(* Logix 5000 project; controller PRU vendor 1 type 14 code 107 rev 20.13; software revision 20.01; part 7 of 17 *)
(* tags used below, declared in another part *)
   DRYER : DUAL_SCREW;
   FAULT : DINT[100];
   FAULT_TIMER : TIMER[10000];
   FAULTS_FA1A_IOK : BOOL;   // MODULE FAULTS ARE OK.
   HMI_ALARM_RESET : BOOL;
   Module_ENCL_Fault : DINT;
   Module_ENCL_Iok : BOOL;
   Module_ENCL_Status : DINT;
   Module_ENCR_Fault : DINT;
   Module_ENCR_Iok : BOOL;
   Module_ENCR_Status : DINT;
   Module_LAI1_Fault : DINT;
   Module_LAI1_Iok : BOOL;
   Module_LAI1_Status : DINT;
   Module_LAI2_Fault : DINT;
   Module_LAI2_Iok : BOOL;
   Module_LAI2_Status : DINT;
   Module_LAI3_Fault : DINT;
   Module_LAI3_Iok : BOOL;
   Module_LAI3_Status : DINT;
   Module_LAO1_Fault : DINT;
   Module_LAO1_Iok : BOOL;
   Module_LAO1_Status : DINT;
   Module_LAO2_Fault : DINT;
   Module_LAO2_Iok : BOOL;
   Module_LAO2_Status : DINT;
   Module_LDI1_Fault : DINT;
   Module_LDI1_Iok : BOOL;
   Module_LDI1_Status : DINT;
   Module_LDI2_Fault : DINT;
   Module_LDI2_Iok : BOOL;
   Module_LDI2_Status : DINT;
   Module_LDO1_Fault : DINT;
   Module_LDO1_Iok : BOOL;
   Module_LDO1_Status : DINT;
   Module_LDO2_Fault : DINT;
   Module_LDO2_Iok : BOOL;
   Module_LDO2_Status : DINT;
   Module_LTC1_Fault : DINT;
   Module_LTC1_Iok : BOOL;
   Module_LTC1_Status : DINT;
   Module_LTC2_Fault : DINT;
   Module_LTC2_Iok : BOOL;
   Module_LTC2_Status : DINT;
   Module_LTC3_Fault : DINT;
   Module_LTC3_Iok : BOOL;
   Module_LTC3_Status : DINT;
   Module_LTC4_Fault : DINT;
   Module_LTC4_Iok : BOOL;
   Module_LTC4_Status : DINT;
   TE0101 : REAL;
   TE0102 : REAL;
   TE0103 : REAL;
   TE0104 : REAL;
   TE0105 : REAL;
   TE0106 : REAL;
   TE0107 : REAL;
   TE0108 : REAL;
   TE0109 : REAL;
   TE0110 : REAL;
   TE0111 : REAL;
   TE0112 : REAL;
   TE0113 : REAL;
   TE0114 : REAL;
   TE0115 : REAL;
   TE0116 : REAL;
   TE0117 : REAL;
   TE0118 : REAL;
   TE0119 : REAL;
   TE0120 : REAL;
   TE0121 : REAL;
   TE0122 : REAL;
   TE0123 : REAL;
   TE0124 : REAL;
   TE0125 : REAL;
   TE0126 : REAL;
   TE0127 : REAL;
   TE0128 : REAL;
   TE0129 : REAL;
   TE0130 : REAL;
   TE0201 : REAL;
   TE0202 : REAL;
   THRESHOLD : REAL[9000];
   WARNF_IOK : BOOL;
   WARNG_IOK : BOOL;
   WEIGHT : REAL;
(* MainProgram, continued *)

ROUTINE B00_WARN_F_700_LO_TEMP   (* ladder *)
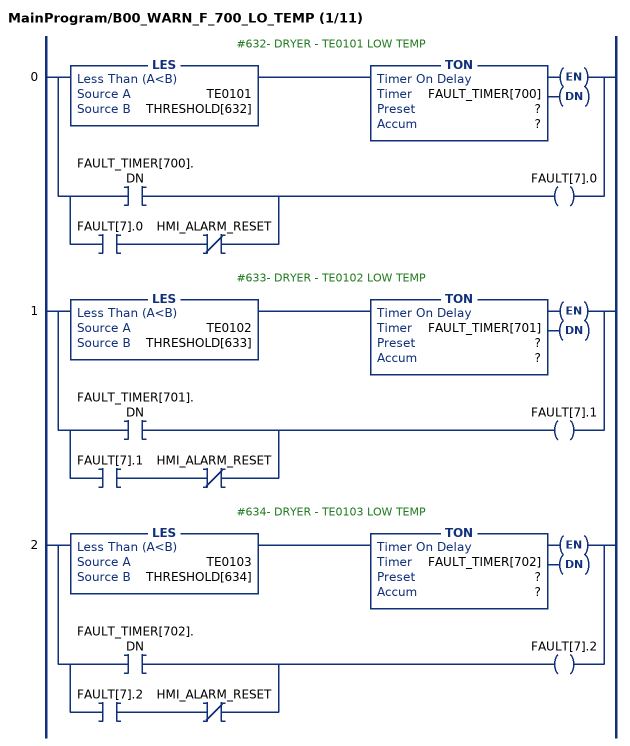
   // #632- DRYER - TE0101 LOW TEMP
   0: [LES(TE0101,THRESHOLD[632]) TON(FAULT_TIMER[700],?,?) ,[XIC(FAULT_TIMER[700].DN) ,XIC(FAULT[7].0) XIO(HMI_ALARM_RESET) ] OTE(FAULT[7].0) ];
   // #633- DRYER - TE0102 LOW TEMP
   1: [LES(TE0102,THRESHOLD[633]) TON(FAULT_TIMER[701],?,?) ,[XIC(FAULT_TIMER[701].DN) ,XIC(FAULT[7].1) XIO(HMI_ALARM_RESET) ] OTE(FAULT[7].1) ];
   // #634- DRYER - TE0103 LOW TEMP
   2: [LES(TE0103,THRESHOLD[634]) TON(FAULT_TIMER[702],?,?) ,[XIC(FAULT_TIMER[702].DN) ,XIC(FAULT[7].2) XIO(HMI_ALARM_RESET) ] OTE(FAULT[7].2) ];
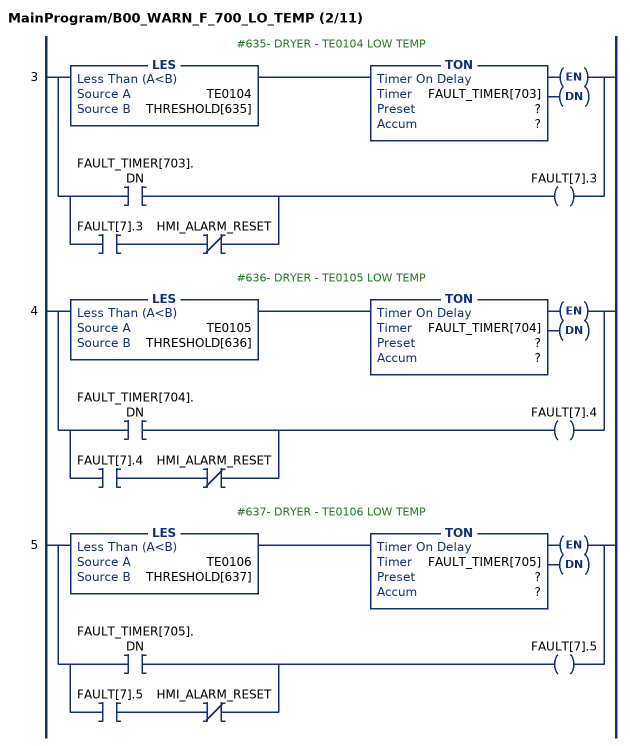
   // #635- DRYER - TE0104 LOW TEMP
   3: [LES(TE0104,THRESHOLD[635]) TON(FAULT_TIMER[703],?,?) ,[XIC(FAULT_TIMER[703].DN) ,XIC(FAULT[7].3) XIO(HMI_ALARM_RESET) ] OTE(FAULT[7].3) ];
   // #636- DRYER - TE0105 LOW TEMP
   4: [LES(TE0105,THRESHOLD[636]) TON(FAULT_TIMER[704],?,?) ,[XIC(FAULT_TIMER[704].DN) ,XIC(FAULT[7].4) XIO(HMI_ALARM_RESET) ] OTE(FAULT[7].4) ];
   // #637- DRYER - TE0106 LOW TEMP
   5: [LES(TE0106,THRESHOLD[637]) TON(FAULT_TIMER[705],?,?) ,[XIC(FAULT_TIMER[705].DN) ,XIC(FAULT[7].5) XIO(HMI_ALARM_RESET) ] OTE(FAULT[7].5) ];
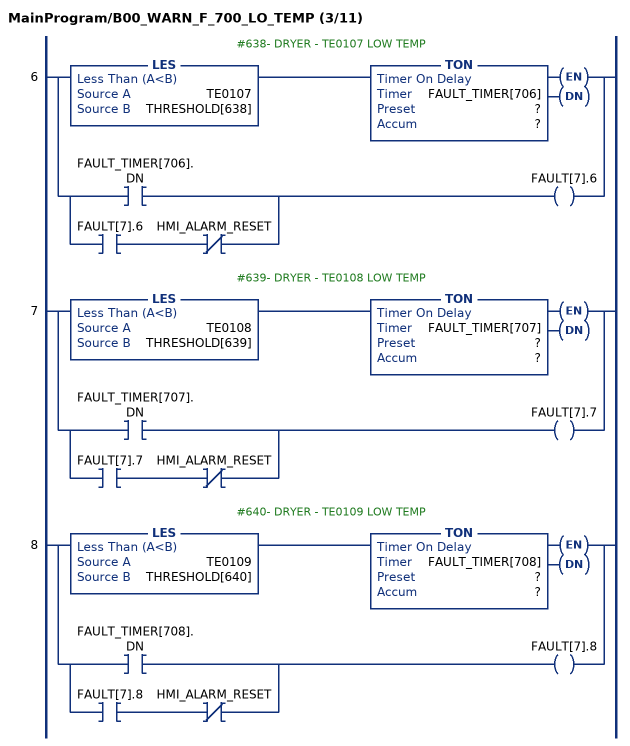
   // #638- DRYER - TE0107 LOW TEMP
   6: [LES(TE0107,THRESHOLD[638]) TON(FAULT_TIMER[706],?,?) ,[XIC(FAULT_TIMER[706].DN) ,XIC(FAULT[7].6) XIO(HMI_ALARM_RESET) ] OTE(FAULT[7].6) ];
   // #639- DRYER - TE0108 LOW TEMP
   7: [LES(TE0108,THRESHOLD[639]) TON(FAULT_TIMER[707],?,?) ,[XIC(FAULT_TIMER[707].DN) ,XIC(FAULT[7].7) XIO(HMI_ALARM_RESET) ] OTE(FAULT[7].7) ];
   // #640- DRYER - TE0109 LOW TEMP
   8: [LES(TE0109,THRESHOLD[640]) TON(FAULT_TIMER[708],?,?) ,[XIC(FAULT_TIMER[708].DN) ,XIC(FAULT[7].8) XIO(HMI_ALARM_RESET) ] OTE(FAULT[7].8) ];
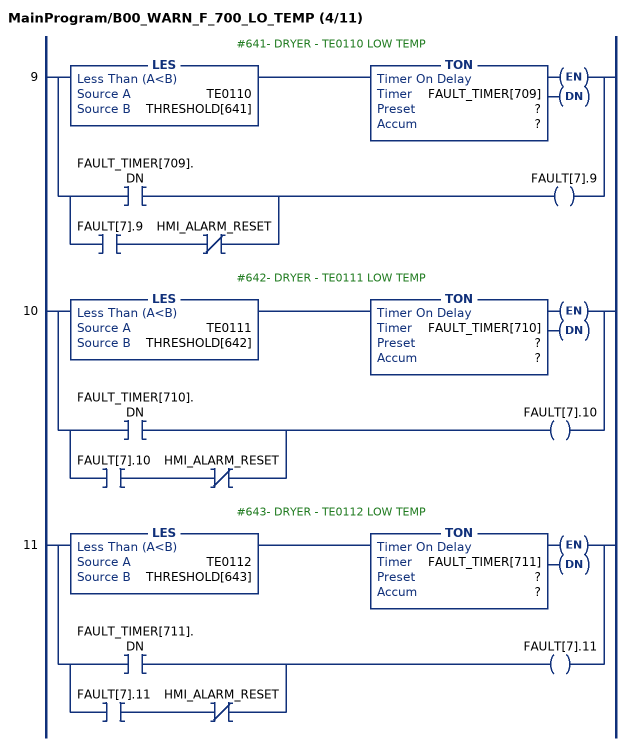
   // #641- DRYER - TE0110 LOW TEMP
   9: [LES(TE0110,THRESHOLD[641]) TON(FAULT_TIMER[709],?,?) ,[XIC(FAULT_TIMER[709].DN) ,XIC(FAULT[7].9) XIO(HMI_ALARM_RESET) ] OTE(FAULT[7].9) ];
   // #642- DRYER - TE0111 LOW TEMP
   10: [LES(TE0111,THRESHOLD[642]) TON(FAULT_TIMER[710],?,?) ,[XIC(FAULT_TIMER[710].DN) ,XIC(FAULT[7].10) XIO(HMI_ALARM_RESET) ] OTE(FAULT[7].10) ];
   // #643- DRYER - TE0112 LOW TEMP
   11: [LES(TE0112,THRESHOLD[643]) TON(FAULT_TIMER[711],?,?) ,[XIC(FAULT_TIMER[711].DN) ,XIC(FAULT[7].11) XIO(HMI_ALARM_RESET) ] OTE(FAULT[7].11) ];
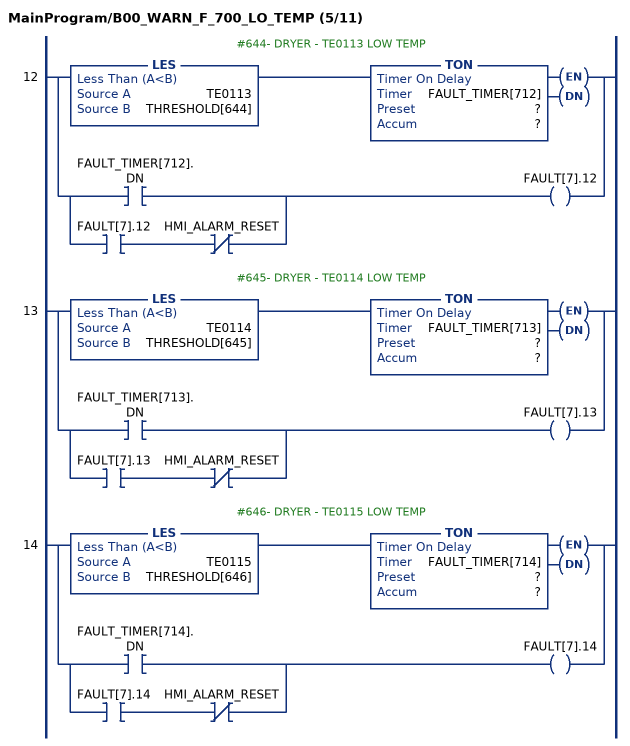
   // #644- DRYER - TE0113 LOW TEMP
   12: [LES(TE0113,THRESHOLD[644]) TON(FAULT_TIMER[712],?,?) ,[XIC(FAULT_TIMER[712].DN) ,XIC(FAULT[7].12) XIO(HMI_ALARM_RESET) ] OTE(FAULT[7].12) ];
   // #645- DRYER - TE0114 LOW TEMP
   13: [LES(TE0114,THRESHOLD[645]) TON(FAULT_TIMER[713],?,?) ,[XIC(FAULT_TIMER[713].DN) ,XIC(FAULT[7].13) XIO(HMI_ALARM_RESET) ] OTE(FAULT[7].13) ];
   // #646- DRYER - TE0115 LOW TEMP
   14: [LES(TE0115,THRESHOLD[646]) TON(FAULT_TIMER[714],?,?) ,[XIC(FAULT_TIMER[714].DN) ,XIC(FAULT[7].14) XIO(HMI_ALARM_RESET) ] OTE(FAULT[7].14) ];
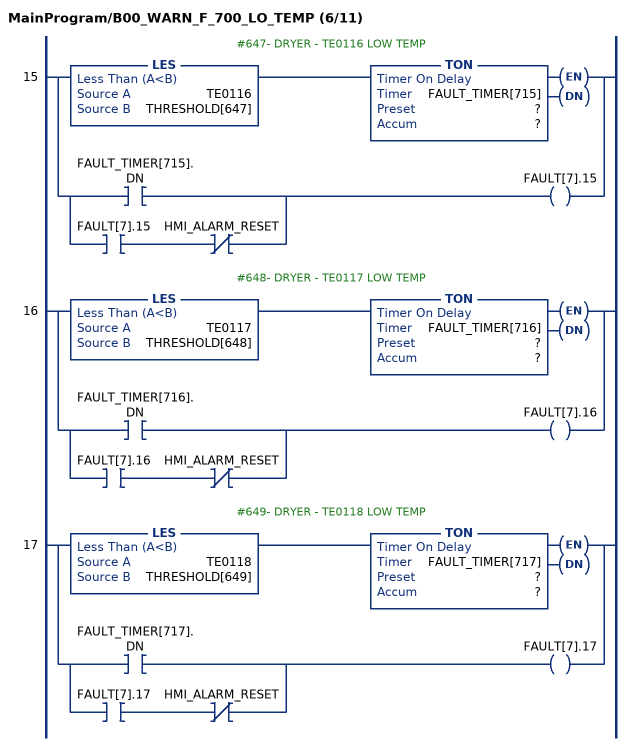
   // #647- DRYER - TE0116 LOW TEMP
   15: [LES(TE0116,THRESHOLD[647]) TON(FAULT_TIMER[715],?,?) ,[XIC(FAULT_TIMER[715].DN) ,XIC(FAULT[7].15) XIO(HMI_ALARM_RESET) ] OTE(FAULT[7].15) ];
   // #648- DRYER - TE0117 LOW TEMP
   16: [LES(TE0117,THRESHOLD[648]) TON(FAULT_TIMER[716],?,?) ,[XIC(FAULT_TIMER[716].DN) ,XIC(FAULT[7].16) XIO(HMI_ALARM_RESET) ] OTE(FAULT[7].16) ];
   // #649- DRYER - TE0118 LOW TEMP
   17: [LES(TE0118,THRESHOLD[649]) TON(FAULT_TIMER[717],?,?) ,[XIC(FAULT_TIMER[717].DN) ,XIC(FAULT[7].17) XIO(HMI_ALARM_RESET) ] OTE(FAULT[7].17) ];
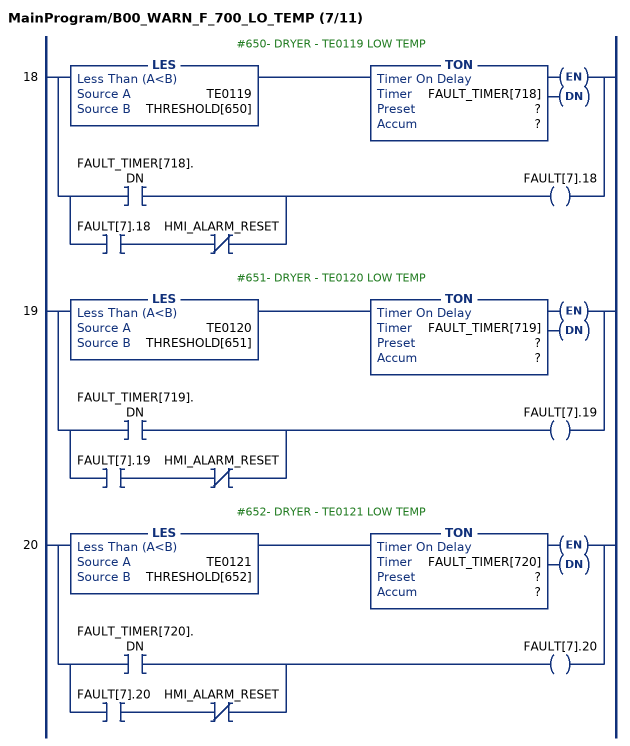
   // #650- DRYER - TE0119 LOW TEMP
   18: [LES(TE0119,THRESHOLD[650]) TON(FAULT_TIMER[718],?,?) ,[XIC(FAULT_TIMER[718].DN) ,XIC(FAULT[7].18) XIO(HMI_ALARM_RESET) ] OTE(FAULT[7].18) ];
   // #651- DRYER - TE0120 LOW TEMP
   19: [LES(TE0120,THRESHOLD[651]) TON(FAULT_TIMER[719],?,?) ,[XIC(FAULT_TIMER[719].DN) ,XIC(FAULT[7].19) XIO(HMI_ALARM_RESET) ] OTE(FAULT[7].19) ];
   // #652- DRYER - TE0121 LOW TEMP
   20: [LES(TE0121,THRESHOLD[652]) TON(FAULT_TIMER[720],?,?) ,[XIC(FAULT_TIMER[720].DN) ,XIC(FAULT[7].20) XIO(HMI_ALARM_RESET) ] OTE(FAULT[7].20) ];
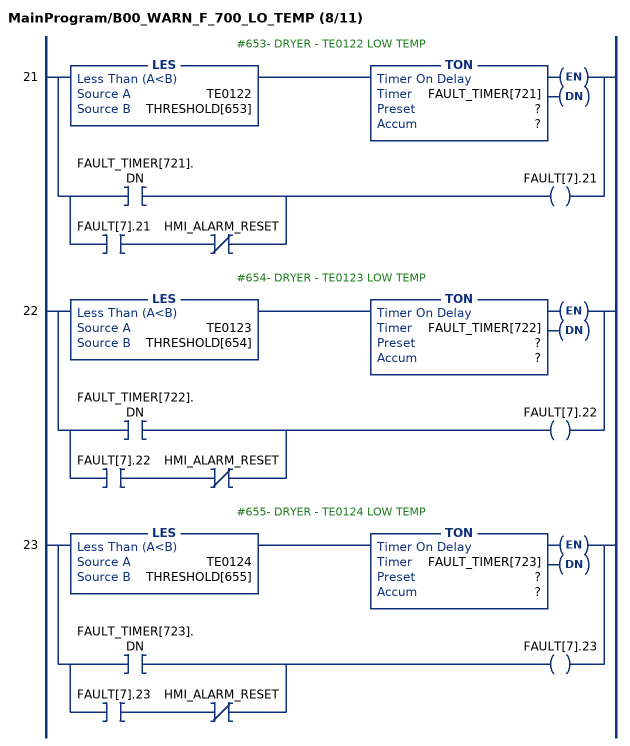
   // #653- DRYER - TE0122 LOW TEMP
   21: [LES(TE0122,THRESHOLD[653]) TON(FAULT_TIMER[721],?,?) ,[XIC(FAULT_TIMER[721].DN) ,XIC(FAULT[7].21) XIO(HMI_ALARM_RESET) ] OTE(FAULT[7].21) ];
   // #654- DRYER - TE0123 LOW TEMP
   22: [LES(TE0123,THRESHOLD[654]) TON(FAULT_TIMER[722],?,?) ,[XIC(FAULT_TIMER[722].DN) ,XIC(FAULT[7].22) XIO(HMI_ALARM_RESET) ] OTE(FAULT[7].22) ];
   // #655- DRYER - TE0124 LOW TEMP
   23: [LES(TE0124,THRESHOLD[655]) TON(FAULT_TIMER[723],?,?) ,[XIC(FAULT_TIMER[723].DN) ,XIC(FAULT[7].23) XIO(HMI_ALARM_RESET) ] OTE(FAULT[7].23) ];
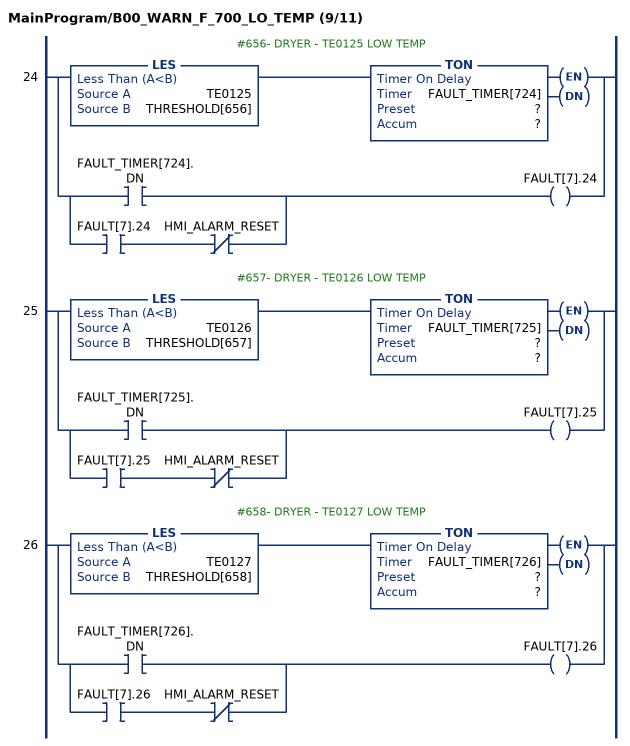
   // #656- DRYER - TE0125 LOW TEMP
   24: [LES(TE0125,THRESHOLD[656]) TON(FAULT_TIMER[724],?,?) ,[XIC(FAULT_TIMER[724].DN) ,XIC(FAULT[7].24) XIO(HMI_ALARM_RESET) ] OTE(FAULT[7].24) ];
   // #657- DRYER - TE0126 LOW TEMP
   25: [LES(TE0126,THRESHOLD[657]) TON(FAULT_TIMER[725],?,?) ,[XIC(FAULT_TIMER[725].DN) ,XIC(FAULT[7].25) XIO(HMI_ALARM_RESET) ] OTE(FAULT[7].25) ];
   // #658- DRYER - TE0127 LOW TEMP
   26: [LES(TE0127,THRESHOLD[658]) TON(FAULT_TIMER[726],?,?) ,[XIC(FAULT_TIMER[726].DN) ,XIC(FAULT[7].26) XIO(HMI_ALARM_RESET) ] OTE(FAULT[7].26) ];
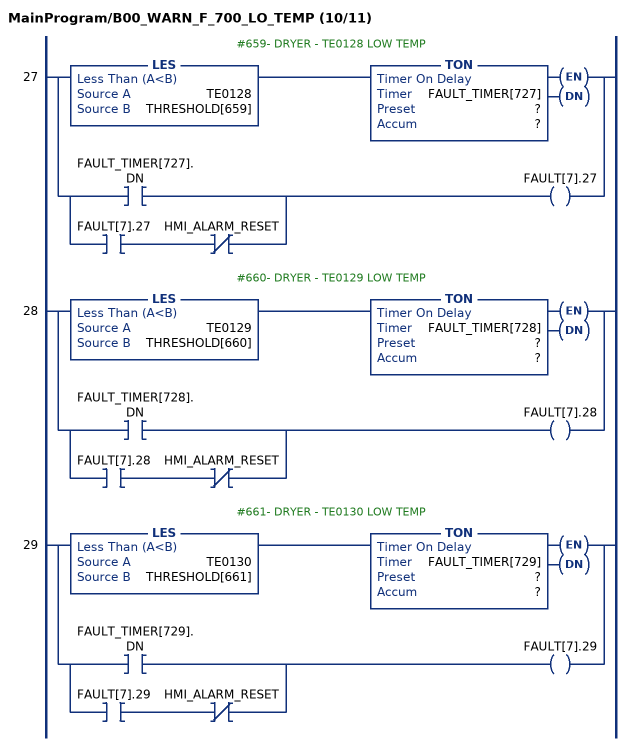
   // #659- DRYER - TE0128 LOW TEMP
   27: [LES(TE0128,THRESHOLD[659]) TON(FAULT_TIMER[727],?,?) ,[XIC(FAULT_TIMER[727].DN) ,XIC(FAULT[7].27) XIO(HMI_ALARM_RESET) ] OTE(FAULT[7].27) ];
   // #660- DRYER - TE0129 LOW TEMP
   28: [LES(TE0129,THRESHOLD[660]) TON(FAULT_TIMER[728],?,?) ,[XIC(FAULT_TIMER[728].DN) ,XIC(FAULT[7].28) XIO(HMI_ALARM_RESET) ] OTE(FAULT[7].28) ];
   // #661- DRYER - TE0130 LOW TEMP
   29: [LES(TE0130,THRESHOLD[661]) TON(FAULT_TIMER[729],?,?) ,[XIC(FAULT_TIMER[729].DN) ,XIC(FAULT[7].29) XIO(HMI_ALARM_RESET) ] OTE(FAULT[7].29) ];
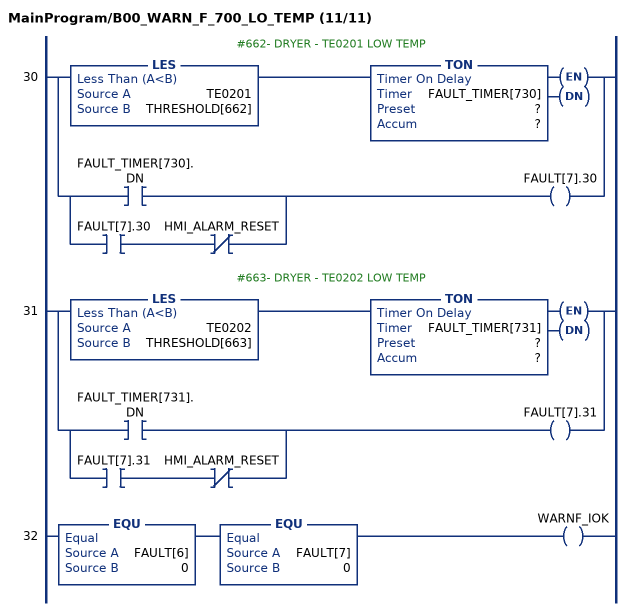
   // #662- DRYER - TE0201 LOW TEMP
   30: [LES(TE0201,THRESHOLD[662]) TON(FAULT_TIMER[730],?,?) ,[XIC(FAULT_TIMER[730].DN) ,XIC(FAULT[7].30) XIO(HMI_ALARM_RESET) ] OTE(FAULT[7].30) ];
   // #663- DRYER - TE0202 LOW TEMP
   31: [LES(TE0202,THRESHOLD[663]) TON(FAULT_TIMER[731],?,?) ,[XIC(FAULT_TIMER[731].DN) ,XIC(FAULT[7].31) XIO(HMI_ALARM_RESET) ] OTE(FAULT[7].31) ];
   32: EQU(FAULT[6],0)EQU(FAULT[7],0)OTE(WARNF_IOK);
END_ROUTINE

ROUTINE B00_WARN_G_800_SCALE   (* ladder *)
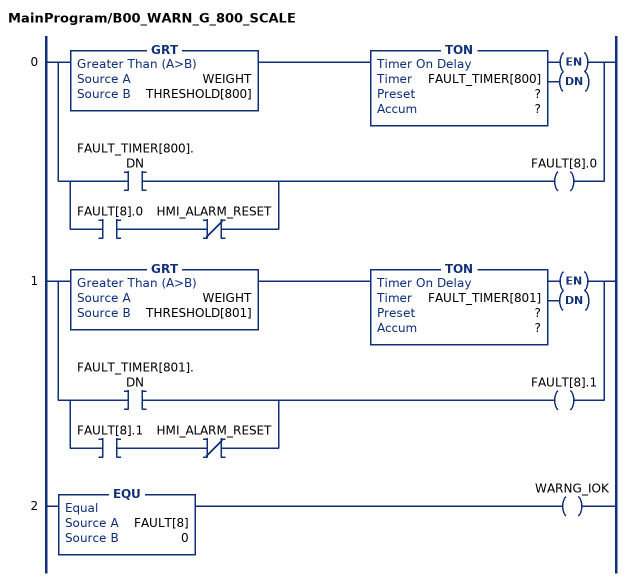
   0: [GRT(WEIGHT,THRESHOLD[800]) TON(FAULT_TIMER[800],?,?) ,[XIC(FAULT_TIMER[800].DN) ,XIC(FAULT[8].0) XIO(HMI_ALARM_RESET) ] OTE(FAULT[8].0) ];
   1: [GRT(WEIGHT,THRESHOLD[801]) TON(FAULT_TIMER[801],?,?) ,[XIC(FAULT_TIMER[801].DN) ,XIC(FAULT[8].1) XIO(HMI_ALARM_RESET) ] OTE(FAULT[8].1) ];
   2: EQU(FAULT[8],0)OTE(WARNG_IOK);
END_ROUTINE

ROUTINE B01_FAULTS_FA1_A_MODULE_1000   (* ladder *)
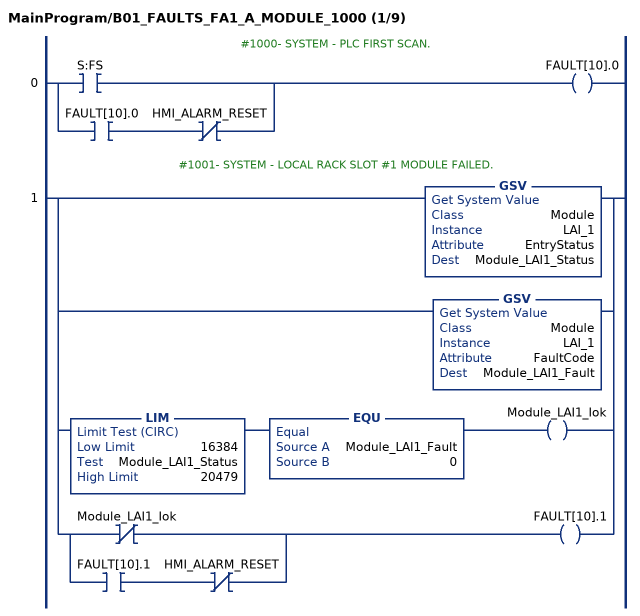
   // #1000- SYSTEM - PLC FIRST SCAN.
   0: [XIC(S:FS) ,XIC(FAULT[10].0) XIO(HMI_ALARM_RESET) ]OTE(FAULT[10].0);
   // #1001- SYSTEM - LOCAL RACK SLOT #1 MODULE FAILED.
   1: [GSV(Module,LAI_1,EntryStatus,Module_LAI1_Status) ,GSV(Module,LAI_1,FaultCode,Module_LAI1_Fault) ,LIM(16384,Module_LAI1_Status,20479) EQU(Module_LAI1_Fault,0) OTE(Module_LAI1_Iok) ,[XIO(Module_LAI1_Iok) ,XIC(FAULT[10].1) XIO(HMI_ALARM_RESET) ] OTE(FAULT[10].1) ];
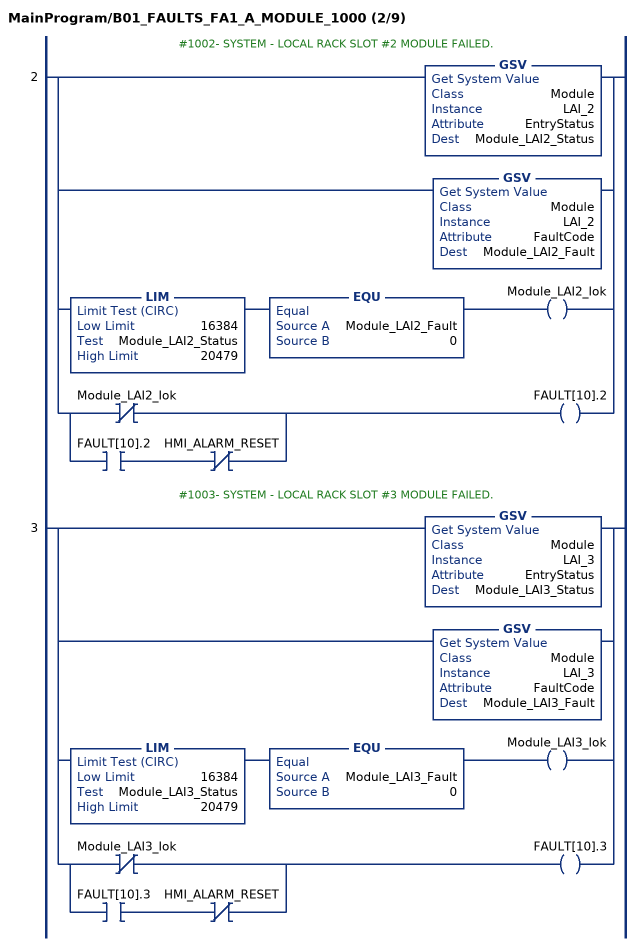
   // #1002- SYSTEM - LOCAL RACK SLOT #2 MODULE FAILED.
   2: [GSV(Module,LAI_2,EntryStatus,Module_LAI2_Status) ,GSV(Module,LAI_2,FaultCode,Module_LAI2_Fault) ,LIM(16384,Module_LAI2_Status,20479) EQU(Module_LAI2_Fault,0) OTE(Module_LAI2_Iok) ,[XIO(Module_LAI2_Iok) ,XIC(FAULT[10].2) XIO(HMI_ALARM_RESET) ] OTE(FAULT[10].2) ];
   // #1003- SYSTEM - LOCAL RACK SLOT #3 MODULE FAILED.
   3: [GSV(Module,LAI_3,EntryStatus,Module_LAI3_Status) ,GSV(Module,LAI_3,FaultCode,Module_LAI3_Fault) ,LIM(16384,Module_LAI3_Status,20479) EQU(Module_LAI3_Fault,0) OTE(Module_LAI3_Iok) ,[XIO(Module_LAI3_Iok) ,XIC(FAULT[10].3) XIO(HMI_ALARM_RESET) ] OTE(FAULT[10].3) ];
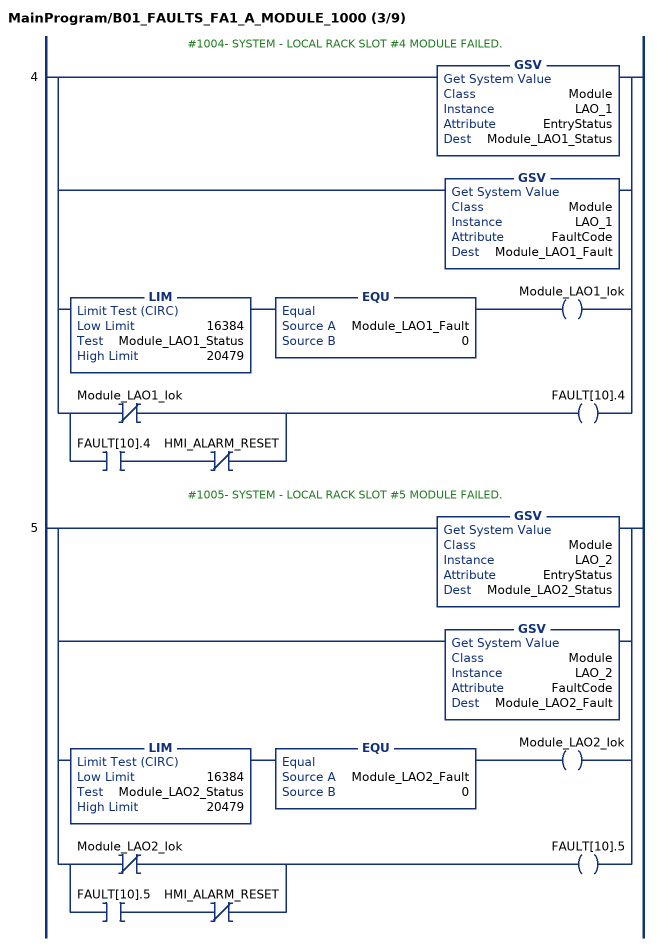
   // #1004- SYSTEM - LOCAL RACK SLOT #4 MODULE FAILED.
   4: [GSV(Module,LAO_1,EntryStatus,Module_LAO1_Status) ,GSV(Module,LAO_1,FaultCode,Module_LAO1_Fault) ,LIM(16384,Module_LAO1_Status,20479) EQU(Module_LAO1_Fault,0) OTE(Module_LAO1_Iok) ,[XIO(Module_LAO1_Iok) ,XIC(FAULT[10].4) XIO(HMI_ALARM_RESET) ] OTE(FAULT[10].4) ];
   // #1005- SYSTEM - LOCAL RACK SLOT #5 MODULE FAILED.
   5: [GSV(Module,LAO_2,EntryStatus,Module_LAO2_Status) ,GSV(Module,LAO_2,FaultCode,Module_LAO2_Fault) ,LIM(16384,Module_LAO2_Status,20479) EQU(Module_LAO2_Fault,0) OTE(Module_LAO2_Iok) ,[XIO(Module_LAO2_Iok) ,XIC(FAULT[10].5) XIO(HMI_ALARM_RESET) ] OTE(FAULT[10].5) ];
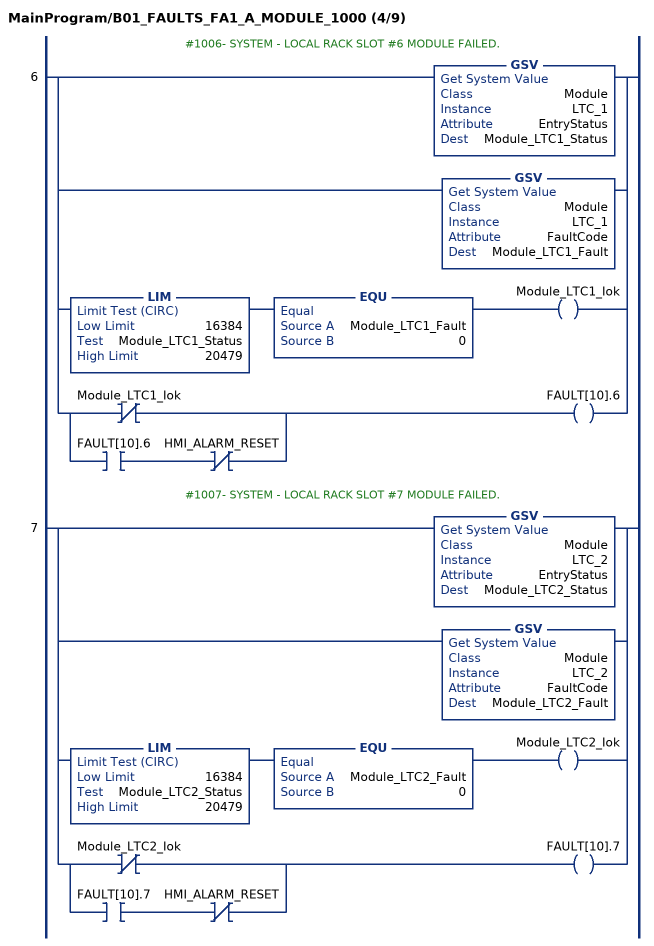
   // #1006- SYSTEM - LOCAL RACK SLOT #6 MODULE FAILED.
   6: [GSV(Module,LTC_1,EntryStatus,Module_LTC1_Status) ,GSV(Module,LTC_1,FaultCode,Module_LTC1_Fault) ,LIM(16384,Module_LTC1_Status,20479) EQU(Module_LTC1_Fault,0) OTE(Module_LTC1_Iok) ,[XIO(Module_LTC1_Iok) ,XIC(FAULT[10].6) XIO(HMI_ALARM_RESET) ] OTE(FAULT[10].6) ];
   // #1007- SYSTEM - LOCAL RACK SLOT #7 MODULE FAILED.
   7: [GSV(Module,LTC_2,EntryStatus,Module_LTC2_Status) ,GSV(Module,LTC_2,FaultCode,Module_LTC2_Fault) ,LIM(16384,Module_LTC2_Status,20479) EQU(Module_LTC2_Fault,0) OTE(Module_LTC2_Iok) ,[XIO(Module_LTC2_Iok) ,XIC(FAULT[10].7) XIO(HMI_ALARM_RESET) ] OTE(FAULT[10].7) ];
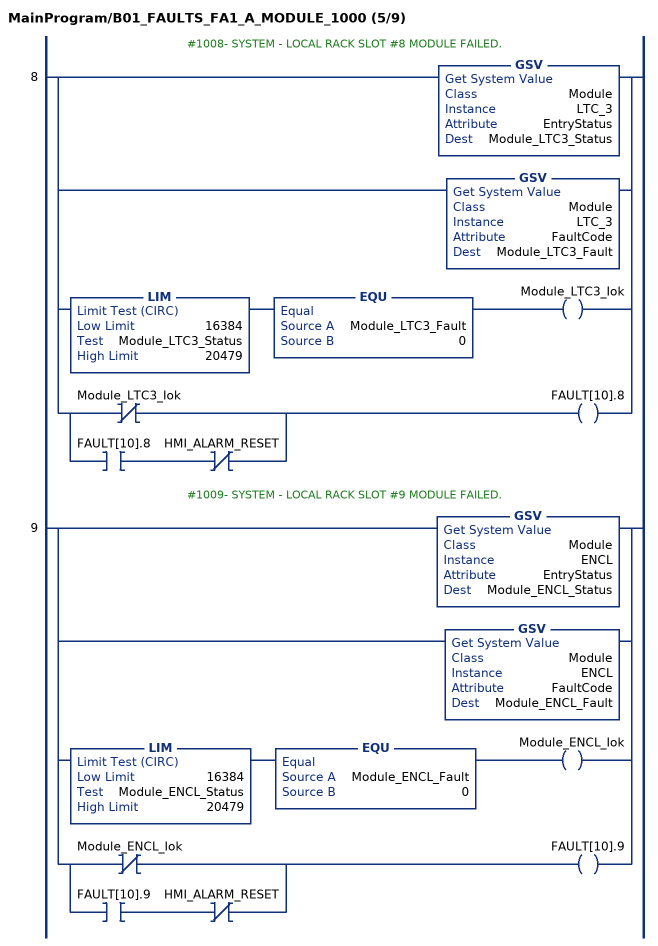
   // #1008- SYSTEM - LOCAL RACK SLOT #8 MODULE FAILED.
   8: [GSV(Module,LTC_3,EntryStatus,Module_LTC3_Status) ,GSV(Module,LTC_3,FaultCode,Module_LTC3_Fault) ,LIM(16384,Module_LTC3_Status,20479) EQU(Module_LTC3_Fault,0) OTE(Module_LTC3_Iok) ,[XIO(Module_LTC3_Iok) ,XIC(FAULT[10].8) XIO(HMI_ALARM_RESET) ] OTE(FAULT[10].8) ];
   // #1009- SYSTEM - LOCAL RACK SLOT #9 MODULE FAILED.
   9: [GSV(Module,ENCL,EntryStatus,Module_ENCL_Status) ,GSV(Module,ENCL,FaultCode,Module_ENCL_Fault) ,LIM(16384,Module_ENCL_Status,20479) EQU(Module_ENCL_Fault,0) OTE(Module_ENCL_Iok) ,[XIO(Module_ENCL_Iok) ,XIC(FAULT[10].9) XIO(HMI_ALARM_RESET) ] OTE(FAULT[10].9) ];
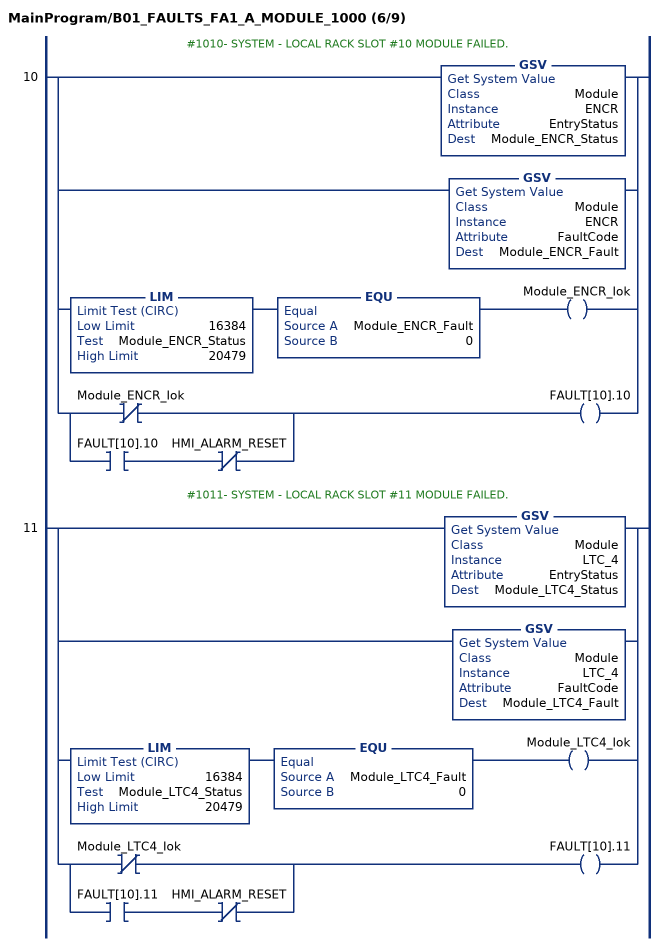
   // #1010- SYSTEM - LOCAL RACK SLOT #10 MODULE FAILED.
   10: [GSV(Module,ENCR,EntryStatus,Module_ENCR_Status) ,GSV(Module,ENCR,FaultCode,Module_ENCR_Fault) ,LIM(16384,Module_ENCR_Status,20479) EQU(Module_ENCR_Fault,0) OTE(Module_ENCR_Iok) ,[XIO(Module_ENCR_Iok) ,XIC(FAULT[10].10) XIO(HMI_ALARM_RESET) ] OTE(FAULT[10].10) ];
   // #1011- SYSTEM - LOCAL RACK SLOT #11 MODULE FAILED.
   11: [GSV(Module,LTC_4,EntryStatus,Module_LTC4_Status) ,GSV(Module,LTC_4,FaultCode,Module_LTC4_Fault) ,LIM(16384,Module_LTC4_Status,20479) EQU(Module_LTC4_Fault,0) OTE(Module_LTC4_Iok) ,[XIO(Module_LTC4_Iok) ,XIC(FAULT[10].11) XIO(HMI_ALARM_RESET) ] OTE(FAULT[10].11) ];
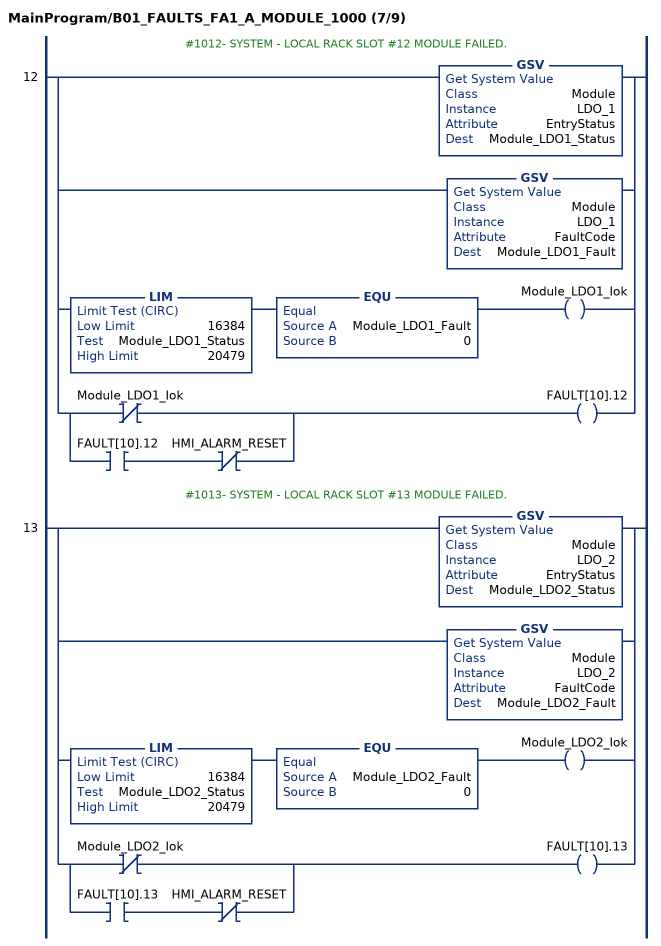
   // #1012- SYSTEM - LOCAL RACK SLOT #12 MODULE FAILED.
   12: [GSV(Module,LDO_1,EntryStatus,Module_LDO1_Status) ,GSV(Module,LDO_1,FaultCode,Module_LDO1_Fault) ,LIM(16384,Module_LDO1_Status,20479) EQU(Module_LDO1_Fault,0) OTE(Module_LDO1_Iok) ,[XIO(Module_LDO1_Iok) ,XIC(FAULT[10].12) XIO(HMI_ALARM_RESET) ] OTE(FAULT[10].12) ];
   // #1013- SYSTEM - LOCAL RACK SLOT #13 MODULE FAILED.
   13: [GSV(Module,LDO_2,EntryStatus,Module_LDO2_Status) ,GSV(Module,LDO_2,FaultCode,Module_LDO2_Fault) ,LIM(16384,Module_LDO2_Status,20479) EQU(Module_LDO2_Fault,0) OTE(Module_LDO2_Iok) ,[XIO(Module_LDO2_Iok) ,XIC(FAULT[10].13) XIO(HMI_ALARM_RESET) ] OTE(FAULT[10].13) ];
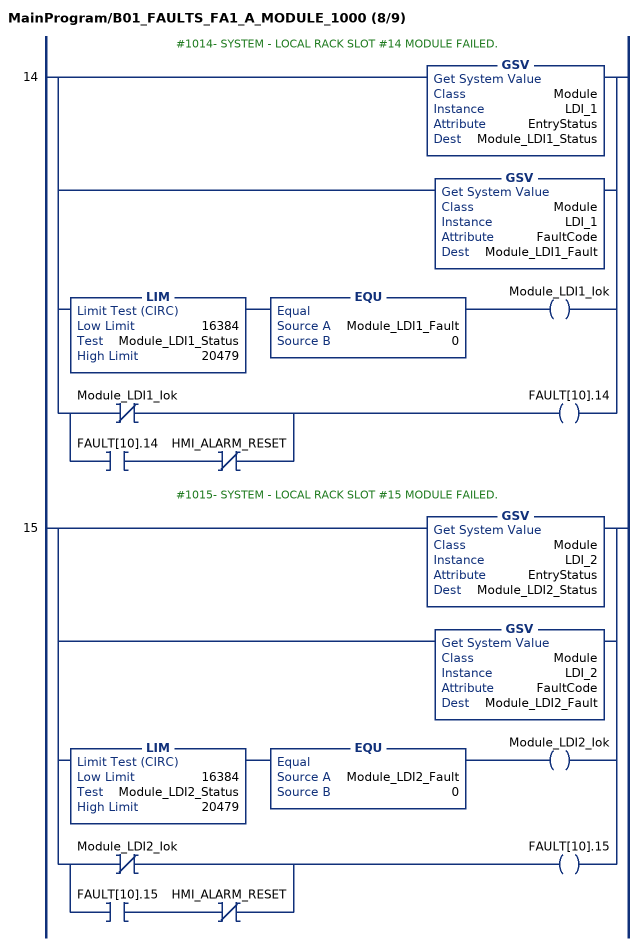
   // #1014- SYSTEM - LOCAL RACK SLOT #14 MODULE FAILED.
   14: [GSV(Module,LDI_1,EntryStatus,Module_LDI1_Status) ,GSV(Module,LDI_1,FaultCode,Module_LDI1_Fault) ,LIM(16384,Module_LDI1_Status,20479) EQU(Module_LDI1_Fault,0) OTE(Module_LDI1_Iok) ,[XIO(Module_LDI1_Iok) ,XIC(FAULT[10].14) XIO(HMI_ALARM_RESET) ] OTE(FAULT[10].14) ];
   // #1015- SYSTEM - LOCAL RACK SLOT #15 MODULE FAILED.
   15: [GSV(Module,LDI_2,EntryStatus,Module_LDI2_Status) ,GSV(Module,LDI_2,FaultCode,Module_LDI2_Fault) ,LIM(16384,Module_LDI2_Status,20479) EQU(Module_LDI2_Fault,0) OTE(Module_LDI2_Iok) ,[XIO(Module_LDI2_Iok) ,XIC(FAULT[10].15) XIO(HMI_ALARM_RESET) ] OTE(FAULT[10].15) ];
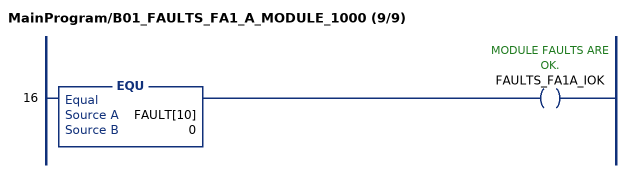
   16: EQU(FAULT[10],0)OTE(FAULTS_FA1A_IOK);
END_ROUTINE
